TYPE AdsTagsParallelUnits :
STRUCT
	Settings: ParallelUnitsSettings;
	Status: ParallelUnitsStatus;
END_STRUCT
END_TYPE

(* stored: Version 1.1.0.1, ProductVersion 3.1.4024.6
   DUT AdsTagsParallelUnits: Id {2f3c55c8-7f85-4e06-bce2-a3e18fdf7c9a} *)
